(* CoDeSys 2.3 export: STUDNIA.EXP *)

(* POU Rooms/Studnia, ST *)
FUNCTION_BLOCK Studnia
VAR_INPUT
END_VAR
VAR_OUTPUT
END_VAR
VAR
END_VAR
D3_4:= D3_1a AND D3_1d;
END_FUNCTION_BLOCK
